KUKA KRL data list: setup_blocks.dat

&ACCESS RV1
&PARAM EDITMASK = *
&PARAM TEMPLATE = C:\KRC\Roboter\Template\ExpertVorgabe
DEFDAT setup_blocks PUBLIC

ENDDAT
